# EPICS substitutions: devel/epics/drivers/v450/v450App/Db/userHost.substitutions
# Example substitutions file

file "db/dbExample1.db" {
    { user = "bonneauHost" }
}

file db/dbExample2.db {
    pattern { user, no, scan }
        { "bonneauHost", 1, "1 second" }
        { "bonneauHost", 2, "2 second" }
        { "bonneauHost", 3, "5 second" }
}
